// TIA Portal project "FactoryIO_Template_S7-1200_V16_V16" (V16)
// Vorlageprojekt für das Buch mit Zielsystem S7-1200

(* hardware
DEVICE "S7-1200-Station_1"  S7-1200 Station
   slot 0: "Baugruppenträger_0"  Rack  V1.0
   slot 1: "PLC_1"  CPU 1211C DC/DC/DC  6ES7 211-1AE40-0XB0  V4.1
*)

// ===== PLC "PLC_1"  CPU 1211C DC/DC/DC =====

VAR_GLOBAL   // PLC tag table "Standard-Variablentabelle"
   "START" AT %I0.0 : Bool;
   "STOP" AT %I0.1 : Bool;
   "SENSOR 1" AT %I0.2 : Bool;
   "SENSOR 2" AT %I0.3 : Bool;
   "SENSOR 3" AT %I0.4 : Bool;
   "MOVING X" AT %I0.6 : Bool;
   "MOVING Z" AT %I0.7 : Bool;
   "DETECTED" AT %I1.0 : Bool;
   "BELT 4m" AT %Q0.0 : Bool;
   "BELT 1 6m" AT %Q0.1 : Bool;
   "BELT 2 6m" AT %Q0.2 : Bool;
   "ROLLER 4m" AT %Q0.3 : Bool;
   "ROLLER 1 6m" AT %Q0.4 : Bool;
   "ROLLER 2 6m" AT %Q0.5 : Bool;
   "X" AT %Q0.6 : Bool;
   "Z" AT %Q0.7 : Bool;
   "GRAB" AT %Q1.0 : Bool;
   "M1" AT %M0.0 : Bool;
   "M2" AT %M0.1 : Bool;
   "M3" AT %M0.2 : Bool;
   "M4" AT %M0.3 : Bool;
   "M5" AT %M0.4 : Bool;
   "M6" AT %M0.5 : Bool;
   "M7" AT %M0.6 : Bool;
   "M8" AT %M0.7 : Bool;
   "M9" AT %M1.0 : Bool;
   "M10" AT %M1.1 : Bool;
   "M11" AT %M1.2 : Bool;
   "M12" AT %M1.3 : Bool;
   "M13" AT %M1.4 : Bool;
   "M14" AT %M1.5 : Bool;
   "M15" AT %M1.6 : Bool;
   "M16" AT %M1.7 : Bool;
END_VAR

FUNCTION "MHJ-PLC-Lab-Function-S71200" : Void   // FC9000, SCL
{ S7_Optimized_Access := 'TRUE' }
VERSION : 0.1
   VAR_TEMP
      rdTimeReturn : Int;
      outputTime : DTL;
      SyncVal : Byte;
      forVal : Int;
      forVal_2 : Int;
      Value : Byte;
   END_VAR
   VAR CONSTANT
      CompVal : Byte := 16#34;
      Value_01 : Byte := 16#11;
      Value_01_DW : DWord := 16#A165_D992;
      Value_02_DW : DWord := 16#58BE_4401;
   END_VAR
BEGIN

   #Value:=PEEK(area := 16#82,
        dbNumber := 0,
        byteOffset := 511);
   #Value := #Value + 1;

   POKE(area := 16#82,
        dbNumber := 0,
        byteOffset := 511,
        value := #Value);

   POKE(area:=16#81,
        dbNumber:=0,
        byteOffset:=1016,
        value:=#Value_01_DW);
   POKE(area := 16#81,
        dbNumber := 0,
        byteOffset := 1020,
        value := #Value_02_DW);

   POKE(area := 16#81,
        dbNumber := 0,
        byteOffset := 511,
        value := B#16#00);

   FOR #forVal := 0 TO 120 DO
       FOR #forVal_2:=0 TO 10 DO
           #rdTimeReturn:=RD_SYS_T(#outputTime);
           #rdTimeReturn := WR_SYS_T(#outputTime);
           #rdTimeReturn := RD_SYS_T(#outputTime);
           #rdTimeReturn := WR_SYS_T(#outputTime);
       END_FOR;
       #SyncVal:= PEEK(area := 16#81,
                      dbNumber := 0,
                      byteOffset := 511);
       IF #SyncVal = #CompVal THEN
          GOTO M_1;
       END_IF;
   END_FOR;
   RETURN;

   M_1:
   POKE(area := 16#81,
        dbNumber := 0,
        byteOffset := 511,
        value := B#16#0);
END_FUNCTION

ORGANIZATION_BLOCK "Main"   // OB1, LAD, ProgramCycle
TITLE = "Main Program Sweep (Cycle)"
{ S7_Optimized_Access := 'TRUE' }
VERSION : 0.1
   VAR_INPUT
      Initial_Call : Bool;   // Initial call of this OB
      Remanence : Bool;   // =True, if remanent data are available
   END_VAR
   VAR_TEMP   // added for the SCL form of the ladder/FBD networks
      _w1 : Bool;
      _w2 : Bool;
      _w3 : Bool;
   END_VAR
BEGIN

REGION Network 1: Konnektierungsbaustein für PLC-Lab
   // Im Netzwerk 1 wird der Konnektierungsbaustein für PLC-Lab aufgerufen.
   // Dieser Aufruf darf nicht entfernt werden!
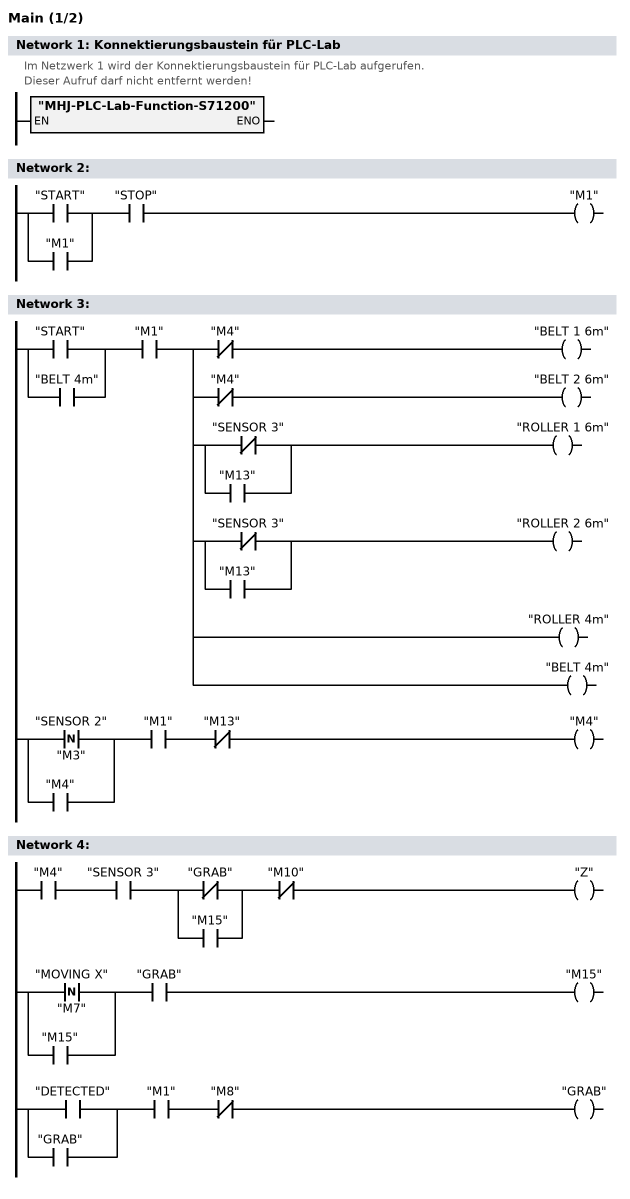
   RUNG wire#powerrail
      "MHJ-PLC-Lab-Function-S71200"()
   END_RUNG
   // the same network as SCL:
   "MHJ-PLC-Lab-Function-S71200"();
END_REGION

REGION Network 2
   RUNG wire#powerrail
      Contact( "START" )
      wire#w1
      Contact( "STOP" )
      Coil( "M1" )
   END_RUNG
   RUNG wire#powerrail
      Contact( "M1" )
   END_RUNG wire#w1
   // the same network as SCL:
   "M1" := ("START" OR "M1") AND "STOP";
END_REGION

REGION Network 3
   RUNG wire#powerrail
      Contact( "START" )
      wire#w1
      Contact( "M1" )
      wire#w2
      I_Contact( "M4" )
      Coil( "BELT 1 6m" )
   END_RUNG
   RUNG wire#powerrail
      Contact( "BELT 4m" )
   END_RUNG wire#w1
   RUNG wire#w2
      I_Contact( "M4" )
      Coil( "BELT 2 6m" )
   END_RUNG
   RUNG wire#w2
      I_Contact( "SENSOR 3" )
      wire#w3
      Coil( "ROLLER 1 6m" )
   END_RUNG
   RUNG wire#w2
      Contact( "M13" )
   END_RUNG wire#w3
   RUNG wire#w2
      I_Contact( "SENSOR 3" )
      wire#w4
      Coil( "ROLLER 2 6m" )
   END_RUNG
   RUNG wire#w2
      Contact( "M13" )
   END_RUNG wire#w4
   RUNG wire#w2
      Coil( "ROLLER 4m" )
   END_RUNG
   RUNG wire#w2
      Coil( "BELT 4m" )
   END_RUNG
   RUNG wire#powerrail
      N_Contact(operand := "SENSOR 2", bit := "M3")
      wire#w5
      Contact( "M1" )
      I_Contact( "M13" )
      Coil( "M4" )
   END_RUNG
   RUNG wire#powerrail
      Contact( "M4" )
   END_RUNG wire#w5
   // the same network as SCL:
   #_w1 := ("START" OR "BELT 4m") AND "M1";
   "BELT 1 6m" := #_w1 AND NOT "M4";
   "BELT 2 6m" := #_w1 AND NOT "M4";
   "ROLLER 1 6m" := #_w1 AND (NOT "SENSOR 3" OR "M13");
   "ROLLER 2 6m" := #_w1 AND (NOT "SENSOR 3" OR "M13");
   "ROLLER 4m" := #_w1;
   "BELT 4m" := #_w1;
   #_w2 := NOT "SENSOR 2" AND "M3";   // falling edge of "SENSOR 2"
   "M3" := "SENSOR 2";
   "M4" := (#_w2 OR "M4") AND "M1" AND NOT "M13";
END_REGION

REGION Network 4
   RUNG wire#powerrail
      Contact( "M4" )
      Contact( "SENSOR 3" )
      wire#w1
      I_Contact( "GRAB" )
      wire#w2
      I_Contact( "M10" )
      Coil( "Z" )
   END_RUNG
   RUNG wire#w1
      Contact( "M15" )
   END_RUNG wire#w2
   RUNG wire#powerrail
      N_Contact(operand := "MOVING X", bit := "M7")
      wire#w3
      Contact( "GRAB" )
      Coil( "M15" )
   END_RUNG
   RUNG wire#powerrail
      Contact( "M15" )
   END_RUNG wire#w3
   RUNG wire#powerrail
      Contact( "DETECTED" )
      wire#w4
      Contact( "M1" )
      I_Contact( "M8" )
      Coil( "GRAB" )
   END_RUNG
   RUNG wire#powerrail
      Contact( "GRAB" )
   END_RUNG wire#w4
   // the same network as SCL:
   "Z" := "M4" AND "SENSOR 3" AND (NOT "GRAB" OR "M15") AND NOT "M10";
   #_w1 := NOT "MOVING X" AND "M7";   // falling edge of "MOVING X"
   "M7" := "MOVING X";
   "M15" := (#_w1 OR "M15") AND "GRAB";
   "GRAB" := ("DETECTED" OR "GRAB") AND "M1" AND NOT "M8";
END_REGION

REGION Network 5
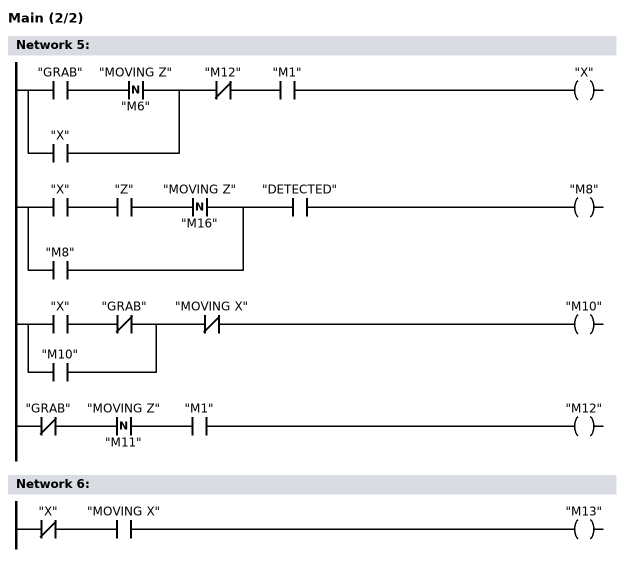
   RUNG wire#powerrail
      Contact( "GRAB" )
      N_Contact(operand := "MOVING Z", bit := "M6")
      wire#w1
      I_Contact( "M12" )
      Contact( "M1" )
      Coil( "X" )
   END_RUNG
   RUNG wire#powerrail
      Contact( "X" )
   END_RUNG wire#w1
   RUNG wire#powerrail
      Contact( "X" )
      Contact( "Z" )
      N_Contact(operand := "MOVING Z", bit := "M16")
      wire#w2
      Contact( "DETECTED" )
      Coil( "M8" )
   END_RUNG
   RUNG wire#powerrail
      Contact( "M8" )
   END_RUNG wire#w2
   RUNG wire#powerrail
      Contact( "X" )
      I_Contact( "GRAB" )
      wire#w3
      I_Contact( "MOVING X" )
      Coil( "M10" )
   END_RUNG
   RUNG wire#powerrail
      Contact( "M10" )
   END_RUNG wire#w3
   RUNG wire#powerrail
      I_Contact( "GRAB" )
      N_Contact(operand := "MOVING Z", bit := "M11")
      Contact( "M1" )
      Coil( "M12" )
   END_RUNG
   // the same network as SCL:
   #_w1 := "GRAB" AND NOT "MOVING Z" AND "M6";   // falling edge of "MOVING Z"
   "M6" := "MOVING Z";
   "X" := (#_w1 OR "X") AND NOT "M12" AND "M1";
   #_w2 := "X" AND "Z" AND NOT "MOVING Z" AND "M16";   // falling edge of "MOVING Z"
   "M16" := "MOVING Z";
   "M8" := (#_w2 OR "M8") AND "DETECTED";
   "M10" := (("X" AND NOT "GRAB") OR "M10") AND NOT "MOVING X";
   #_w3 := NOT "GRAB" AND NOT "MOVING Z" AND "M11";   // falling edge of "MOVING Z"
   "M11" := "MOVING Z";
   "M12" := #_w3 AND "M1";
END_REGION

REGION Network 6
   RUNG wire#powerrail
      I_Contact( "X" )
      Contact( "MOVING X" )
      Coil( "M13" )
   END_RUNG
   // the same network as SCL:
   "M13" := NOT "X" AND "MOVING X";
END_REGION
END_ORGANIZATION_BLOCK